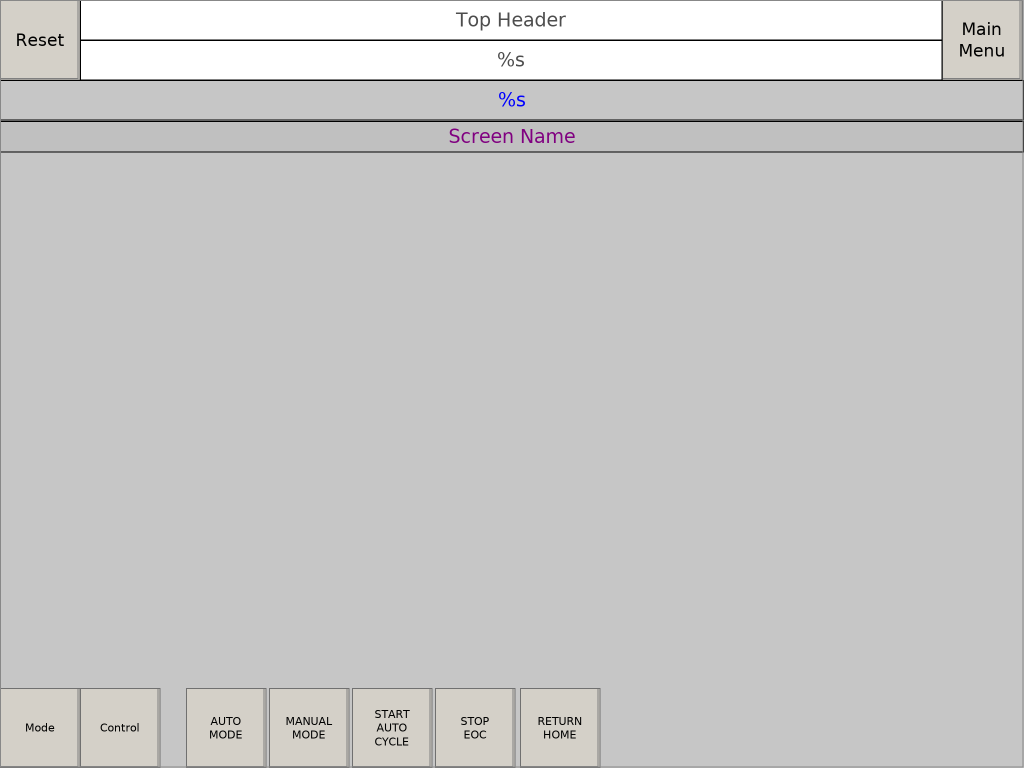
VISUALIZATION SS_91_Template  // 1024x768
    Button (0,0 80x80), "Reset"
    Button (942,0 80x80), "Main Menu"
        OnMouseClick: change screen: SS_10_MenuScreen
    Rectangle (0,80 1024x40), "%s", text variable: GlobalMessages.gMsgMc.Prompts.topMessage, invisible if: HMIData.gHideDisplayElementPromptView.McEnabled, text list: 'Mc_Prompts', text index: HMIData.gNumActivePromptTextList[0]
    Rectangle (80,0 862x40), "Top Header"
    Button (0,688 80x80), "Mode"
        OnMouseClick: change screen: SS_01_ModeScreen
    Rectangle (80,40 862x40), "%s", text variable: GlobalMessages.gMsgMc.Warning.topMessage, invisible if: HMIData.gHideDisplayElementWarningView.McEnabled
    Rectangle (80,40 862x40), "%s", text variable: GlobalMessages.gMsgS1.Warning.topMessage, invisible if: HMIData.gHideDisplayElementWarningView.S1Enabled
    Rectangle (80,40 862x40), "%s", text variable: GlobalMessages.gMsgS2.Warning.topMessage, invisible if: HMIData.gHideDisplayElementWarningView.S2Enabled
    Rectangle (80,40 862x40), "%s", text variable: GlobalMessages.gMsgS3.Warning.topMessage, invisible if: HMIData.gHideDisplayElementWarningView.S3Enabled
    Rectangle (80,40 862x40), "%s", text variable: GlobalMessages.gMsgS4.Warning.topMessage, invisible if: HMIData.gHideDisplayElementWarningView.S4Enabled
    Rectangle (80,40 862x40), "%s", text variable: GlobalMessages.gMsgS5.Warning.topMessage, invisible if: HMIData.gHideDisplayElementWarningView.S5Enabled
    Rectangle (80,40 862x40), "%s", text variable: GlobalMessages.gMsgS6.Warning.topMessage, invisible if: HMIData.gHideDisplayElementWarningView.S6Enabled
    Rectangle (80,40 862x40), "%s", text variable: GlobalMessages.gMsgMc.Alarm.topMessage, invisible if: HMIData.gHideDisplayElementAlarmView.McEnabled
    Rectangle (80,40 862x40), "%s", text variable: GlobalMessages.gMsgS1.Alarm.topMessage, invisible if: HMIData.gHideDisplayElementAlarmView.S1Enabled, text list: ''
    Rectangle (80,40 862x40), "%s", text variable: GlobalMessages.gMsgS2.Alarm.topMessage, invisible if: HMIData.gHideDisplayElementAlarmView.S2Enabled
    Rectangle (80,40 862x40), "%s", text variable: GlobalMessages.gMsgS3.Alarm.topMessage, invisible if: HMIData.gHideDisplayElementAlarmView.S3Enabled
    Rectangle (80,40 862x40), "%s", text variable: GlobalMessages.gMsgS4.Alarm.topMessage, invisible if: HMIData.gHideDisplayElementAlarmView.S4Enabled
    Rectangle (80,40 862x40), "%s", text variable: GlobalMessages.gMsgS5.Alarm.topMessage, invisible if: HMIData.gHideDisplayElementAlarmView.S5Enabled
    Rectangle (80,40 862x40), "%s", text variable: GlobalMessages.gMsgS6.Alarm.topMessage, invisible if: HMIData.gHideDisplayElementAlarmView.S6Enabled
    Rectangle (0,80 1024x40), "%s", text variable: GlobalMessages.gMsgS1.Prompts.topMessage, invisible if: HMIData.gHideDisplayElementPromptView.S1Enabled
    Rectangle (0,80 1024x40), "%s", text variable: GlobalMessages.gMsgS2.Prompts.topMessage, invisible if: HMIData.gHideDisplayElementPromptView.S2Enabled
    Rectangle (0,80 1024x40), "%s", text variable: GlobalMessages.gMsgS3.Prompts.topMessage, invisible if: HMIData.gHideDisplayElementPromptView.S3Enabled
    Rectangle (0,80 1024x40), "%s", text variable: GlobalMessages.gMsgS4.Prompts.topMessage, invisible if: HMIData.gHideDisplayElementPromptView.S4Enabled
    Rectangle (0,80 1024x40), "%s", text variable: GlobalMessages.gMsgS5.Prompts.topMessage, invisible if: HMIData.gHideDisplayElementPromptView.S5Enabled
    Rectangle (0,80 1024x40), "%s", text variable: GlobalMessages.gMsgS6.Prompts.topMessage, invisible if: HMIData.gHideDisplayElementPromptView.S6Enabled
    Rectangle (0,121 1024x31), "Screen Name", invisible if: HMIData.gHideDisplayElementPromptView.S6Enabled, text list: 'ScreenNames', text index: HMIData.gScreenNumber
    Button (80,688 80x80), "Control"
    Button (186,688 80x80), "AUTO MODE", colour toggle: HMIData.btnFdbk.btn00Fdbk
        tap HMIData.btnMode.btnFooterAutoMode
    Button (269,688 80x80), "MANUAL MODE", colour toggle: HMIData.btnFdbk.btn01Fdbk
        tap HMIData.btnMode.btnFooterManualMode
    Button (352,688 80x80), "START AUTO CYCLE", colour toggle: HMIData.btnFdbk.btnAutoCyclingFdbk
        tap HMIData.btnMode.btnFooterAutoCycleStart
    Button (435,688 80x80), "STOP EOC"
        tap HMIData.btnMode.btnFooterAutoCycleStopEOC
    Button (520,688 80x80), "RETURN HOME", colour toggle: HMIData.btnFdbk.btnIsHomeFdbk
        tap HMIData.btnMode.btnFooterReturnHome
END_VISUALIZATION

(* stored: Version 1.1.0.1, ProductVersion 3.1.4024.12
   Visu SS_91_Template: Id {b17fde76-284b-401f-89cc-43a3764876ae} *)
